Staubli VAL3: io.dtx

public sio IOC = {link=Socket\MFX}
dio COLLISIONSENSOR
